(* IEC 61131-3 sources: AXOpen/src/components.drives/app/src/Documentation/TypesStructuresAndEnums, 2 files *)

(* ---- AxoDrive_Data_Example.st ---- *)
NAMESPACE AXOpen.Components.Drives
    {S7.extern=ReadWrite}
    CLASS AxoDrive_Data_Example
        VAR PUBLIC
            Cycle                       :   ULINT;
            OverrideVelocityFactor		:	LREAL := 1.0;	//LREAL value to be written
            OverrideAccelerationFactor	:	LREAL := 1.0;	//LREAL value to be written
            OverrideJerkFactor			:	LREAL := 1.0;	//LREAL value to be written
        END_VAR
    END_CLASS
END_NAMESPACE

(* ---- AxoDrive_Status_Example.st ---- *)
NAMESPACE AXOpen.Components.Drives
    {S7.extern=ReadWrite}
    {#ix-attr:[Container(Layout.Tabs)]}
    CLASS PUBLIC AxoDrive_Status_Example
        VAR PUBLIC
            {#ix-set:AttributeName = "<#DriveStatusWord#>"}
            DriveStatusWord : WORD;
            {#ix-set:AttributeName = "<#ActualPosition#>"}
            ActualPosition : DINT;
            {#ix-set:AttributeName = "<#ActualVelocity#>"}
            ActualVelocity : DINT;
            {#ix-set:AttributeName = "<#DiagnosticMessage#>"}
            DiagnosticMessage : DWORD;
            {#ix-set:AttributeName = "<#ActualTorque#>"}
            ActualTorque : INT;
        END_VAR
    END_CLASS
END_NAMESPACE
